TYPE D_InputVar :
STRUCT
	INT_Var : INT; // Integer input
	Real_Var : REAL; //# 
END_STRUCT
END_TYPE

(* stored: Version 1.1.0.1, ProductVersion 3.1.4024.3
   DUT D_InputVar: Id {f8e5ff37-9e8f-41a4-a552-bdcea736ca42} *)
